FUNCTION_BLOCK DigitalOutputLatched
VAR_INPUT
	on					: BOOL;
	off					: BOOL;
END_VAR
VAR_OUTPUT
	output				: BOOL;
END_VAR

IF off		THEN
	output 	:= FALSE;
ELSIF on 	THEN
	output 	:= TRUE;
END_IF

END_FUNCTION_BLOCK

(* stored: Version 1.1.0.1
   POU DigitalOutputLatched: Id {2714d9d5-4d1f-461b-b06d-603b4874e350}, SpecialFunc None *)
